// TIA Portal V18 export
// export: Created 2026-06-08T03:54:35.444588Z, ExportSetting WithDefaults, DisplayName Totally Integrated Automation Portal, DisplayVersion V18, DisplayName TIA Portal Openness, DisplayVersion V18, DisplayName TIA Portal Version Control Interface, DisplayVersion V18, DisplayName STEP 7 Professional, DisplayVersion V18, DisplayName STEP 7 Safety, DisplayVersion V18, DisplayName WinCC Professional, DisplayVersion V18
FUNCTION "FC_MB_SERVER_COMPAT_TEST" : Void   // FC1, LAD
{ S7_Optimized_Access := 'TRUE' }
VERSION : 0.1
// stored: AutoNumber true, IsIECCheckEnabled false, SetENOAutomatically false, UDAEnableTagReadback false
BEGIN

REGION Network 1
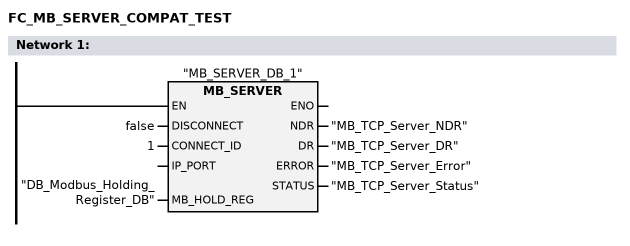
   RUNG wire#powerrail
      { S7_Templates := "[card1200 := 1, card1500 := 0]" } "MB_SERVER_DB_1".MB_SERVER(DISCONNECT := false, CONNECT_ID := 1, IP_PORT :=, MB_HOLD_REG := "DB_Modbus_Holding_Register_DB", NDR => "MB_TCP_Server_NDR", DR => "MB_TCP_Server_DR", ERROR => "MB_TCP_Server_Error", STATUS => "MB_TCP_Server_Status")
   END_RUNG
   // the same network as SCL:
   "MB_SERVER_DB_1"(DISCONNECT := false,   // MB_SERVER
                    CONNECT_ID := 1,
                    MB_HOLD_REG := "DB_Modbus_Holding_Register_DB",
                    NDR => "MB_TCP_Server_NDR",
                    DR => "MB_TCP_Server_DR",
                    ERROR => "MB_TCP_Server_Error",
                    STATUS => "MB_TCP_Server_Status");
END_REGION
END_FUNCTION
